{attribute 'qualified_only'}
// LREAL: Long Real decimal number

VAR_GLOBAL
	
	// Unfiltered Pressures
	fPa 				: LREAL; 	// [bar], Pressure A 
	fPb 				: LREAL; 	// [bar], Pressure B 
	fPs 				: LREAL; 	// [bar], Pressure Supply 
	fPaLower 			: LREAL; 	// [bar], Pressure A between DCV and CBV 
	
	// Filtered Pressures
	fPaFiltered 		: LREAL; 	// [bar], Pressure A Filtered 
	fPbFiltered 		: LREAL; 	// [bar], Pressure B Filtered
	fPsFiltered 		: LREAL; 	// [bar], Pressure Supply Filtered
	fPaLowerFiltered 	: LREAL; 	// [bar], Pressure A between DCV and CBV Filtered
	
	fSpoolPosition 		: LREAL; 	// [-1,1], Spool position
	fPistonPosition 	: LREAL; 	// [m], Piston position
	fPistonPosMeasured 	: LREAL; 	// [m], Measured piston position
	fJoystick 			: LREAL; 	// [-1,1], Joystick signal
	fFlow 				: LREAL; 	// [L/min], Flow rod-side 
	fFlowCalc 			: LREAL; 	// [L/min], Calculated flow
	
	fXRef 				: LREAL; 	// [m], Position reference [m]
	fXDotRef 			: LREAL; 	// [m/s], Velocity reference [m/s]
	fFlowRef 			: LREAL; 	// [L/min], Flow reference calculated form fXDotRef
	
	fFFFlow				: LREAL;	// [L/min], Flow form feed forward
	fKv					: LREAL; 	// [L/min / bar^0.5] K value 

	fWantedSpoolPos 	: LREAL; 	// [-1,1], Wanted spool position
	fUpfbGrad 			: LREAL; 	// Pressure feedback gradient
	fPxGrad 			: LREAL; 	// Pressure gradient
	fUTest 				: LREAL; 	// [-1,1], Signal to Valve with pfb (pressure feedback)
	fTime 				: LREAL; 	// [s], Time
	fError 				: LREAL; 	// [m], Error
	
	
	fSignalPID 			: LREAL; 	// PID signal value
	fFF 				: LREAL; 	// FF signal Value
	fUpfb 				: LREAL; 	// Pressure feedback signal
	fU 					: LREAL; 	// [-1,1], Signal to set spool at wanted position 

END_VAR

(* stored: Version 1.1.0.1
   GVL G_OPC: Id {5ea6be42-d96d-412e-8945-28bb945cf324} *)
